FUNCTION_BLOCK XtsHardwareTestSuite
VAR
	XtsIoEnvVar : XTSIOEnvVarWrapper;
	MyXtsHardware : XTSHardware;
	ReRun: BOOL;
END_VAR

HardwareRejectsCallsWithNoXPU_Test();
HardwareIdentifiesNoXpu_Test();
RegisterXPU_Test();
HardwareWontCycleWithoutInit_Test();
IF ReRun THEN
	TestSuite.ReRunTests();
	ReRun := FALSE;
END_IF

METHOD HardwareIdentifiesNoXpu_Test : BOOL
VAR_INST
	Expected : BOOL := FALSE;
	Actual	 : BOOL;
END_VAR
IF TestSuite.Test(__POUNAME()).ExecuteTest() THEN
	Actual := MyXtsHardware.HasXPU();
	TestSuite.Test(__POUNAME()).AssertEqual(Expected, Actual);
END_IF
END_METHOD

METHOD HardwareRejectsCallsWithNoXPU_Test : BOOL
VAR_INST
	Expected : BOOL := TRUE;
	Actual	 : BOOL;
END_VAR
IF TestSuite.Test(__POUNAME()).ExecuteTest() THEN
	Actual := FAILED(MyXtsHardware.Initialise());
	TestSuite.Test(__POUNAME()).AssertEqual(Expected, Actual);
END_IF
END_METHOD

METHOD HardwareWontCycleWithoutInit_Test : BOOL
VAR_INST
	Expected : BOOL := TRUE;
	Actual	 : BOOL;
END_VAR
IF TestSuite.Test(__POUNAME()).ExecuteTest() THEN
	Actual := FAILED(MyXtsHardware.Cycle());
	TestSuite.Test(__POUNAME()).AssertEqual(Expected, Actual);
END_IF
END_METHOD

METHOD RegisterXPU_Test : BOOL
VAR_INST
	Expected : BOOL := TRUE;
	Actual	 : BOOL;
END_VAR
IF TestSuite.Test(__POUNAME()).ExecuteTest() THEN
	MyXtsHardware.MyXtsIoEnvVarWrapper := XtsIoEnvVar;
	Actual := MyXtsHardware.HasXPU();
	TestSuite.Test(__POUNAME()).AssertEqual(Expected, Actual);
END_IF
END_METHOD

END_FUNCTION_BLOCK

(* stored: Version 1.1.0.1
   POU XtsHardwareTestSuite: Id {b560ca6a-e691-471a-a25d-3f29414ba80e}, SpecialFunc None
   Method HardwareIdentifiesNoXpu_Test: Id {8917a178-edef-4eb2-9cd2-49d29f8c1ec8}
   Method HardwareRejectsCallsWithNoXPU_Test: Id {1788fe5c-f52a-4593-9903-c640bbecef8a}
   Method HardwareWontCycleWithoutInit_Test: Id {fba77493-9432-4925-a6b5-53c91b6f648a}
   Method RegisterXPU_Test: Id {b248b030-f2bc-411a-8466-8dc5754b8803} *)
